FUNCTION_BLOCK TESTPAR_FBD (* Test Java generation of parameters in FBD algorithm *)
  (* Standard: 61499-2 *)
  (* Version 0.1, 2007-11-11, JHC, Holobloc Inc, Deleted import, made a SimpleFB.. *)
  (* Version 0.0, 2004-12-15, JHC, Rockwell Automation *)
  (* Compiler header: package fb.rt.test; *)
  (* Compiler classdef: SimpleFB *)
  (* Compiler Java Sun JDK 1.6.0 *)
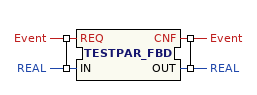
  EVENT_INPUT
    REQ WITH IN; (* Normal Execution Request *)
  END_EVENT
  EVENT_OUTPUT
    CNF WITH OUT; (* Execution Confirmation *)
  END_EVENT
  VAR_INPUT
    IN : REAL;
  END_VAR
  VAR_OUTPUT
    OUT : REAL; (* IN + 2.0 *)
  END_VAR
  ALGORITHM REQ IN FBD: (* Normally executed algorithm *)
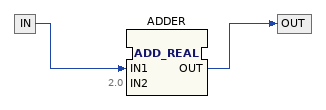
    FBS
      ADDER : ADD_REAL(IN2 := 2.0 (* The parameter *));
    END_FBS
    DATA_CONNECTIONS
      IN TO ADDER.IN1;
      ADDER.OUT TO OUT;
    END_CONNECTIONS
  END_ALGORITHM
END_FUNCTION_BLOCK
